TYPE PTOTargetChannel :
STRUCT
	{attribute addProperty Name "Target counter value"}
	TargetCounterValue AT %Q* : UDINT;
END_STRUCT
END_TYPE

(* stored: Version 1.1.0.1, ProductVersion 3.1.4024.9
   DUT PTOTargetChannel: Id {1b710e62-3dfd-0f39-31cf-77621d4c13ec} *)
